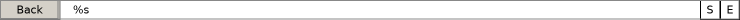
VISUALIZATION VISU_Base_Header  // 740x20
    Button (0,0 60x20), "Back"
        OnMouseClick: change screen: Previous 
    Rectangle (70,0 150x20), "%s", text variable: PRG_SYSTEM.aCurrentDateTime
    RoundedRectangle (700,0 20x20), "S", tooltip "Sleep active", colour toggle: PRG_MACHINE.sO_SystemCmd.bSleep
    RoundedRectangle (720,0 20x20), "E", tooltip "EmergencyStop active", colour toggle: PRG_MACHINE.sO_SystemCmd.bEStop
END_VISUALIZATION

(* stored: Version 1.1.0.1, ProductVersion 3.1.4024.3
   Visu VISU_Base_Header: Id {2855f497-8ce1-47cc-ac01-c570391d34e2} *)
